// TIA Portal V20 export
// export: Created 2025-12-01T14:57:05.6941623Z, ExportSetting None, DisplayName Totally Integrated Automation Portal, DisplayVersion V20 Update 3, DisplayName TIA Portal Openness, DisplayVersion V20 Update 3, DisplayName TIA Portal Version Control Interface, DisplayVersion V20 Update 3, DisplayName STEP 7 Professional, DisplayVersion V20 Update 3, DisplayName STEP 7 Safety, DisplayVersion V20 Update 2, DisplayName WinCC Basic/Comfort/Advanced, DisplayVersion V20 Update 3, DisplayName WinCC Professional, DisplayVersion V20 Update 3, DisplayName WinCC Unified, DisplayVersion V20 Update 3
FUNCTION "FC876_BorrarEstructura" : Void   // FC876, LAD
TITLE = BorrarEstructura
{ S7_Optimized_Access := 'FALSE' }
AUTHOR : TRACKING
NAME : 20130301
VERSION : 3.0
// Borra un numero de bytes de un DB desde Offset que se indique
// stored: AutoNumber false, SetENOAutomatically false
   VAR_INPUT
      NumDB : Word;   // Numero del DB
      POffset : DWord;   // Puntero del Offset dento del DB
      NumBytes : UInt;   // Numero de Bytes que hay que borrar
   END_VAR
   VAR_TEMP
      Guardar_AR1 : DWord;
      Guardar_AR2 : DWord;
      PAny_DB : Any;
      ReturnValor : Int;
      Cero : Byte;
   END_VAR
BEGIN

NETWORK
TITLE = Inicializar Punteros Any
//////////////////////////////////////////////////////////////////////////////
//////////////////////////////////////////////////////////////////////////////
/// Tareas Iniciales

      TAR1  #Guardar_AR1;  // Guardar AR1 y AR2
      TAR2  #Guardar_AR2;


//////////////////////////////////////////////////////////////////////////////
//////////////////////////////////////////////////////////////////////////////
/// Puntero Any Origen

      LAR2  P##PAny_DB;  // - Any - DB de Origen
      L     B#16#10;  //   10H para S7
      T     LB [AR2, P#0.0];
      L     B#16#2;  //   Tipo de Datos (BYTE)
      T     LB [AR2, P#1.0];
      L     #NumBytes;  //   Cantidad de datos
      T     LW [AR2, P#2.0];
      L     #NumDB;  //   Numero de DB
      T     LW [AR2, P#4.0];
      L     #POffset;  //   Direccion de Inicio
      T     LD [AR2, P#6.0];
      L     B#16#84;  //   El Area de Memoria = DB (Nota: No 84)
      T     LB [AR2, P#6.0];


//////////////////////////////////////////////////////////////////////////////
//////////////////////////////////////////////////////////////////////////////
/// Tareas Finales

      LAR1  #Guardar_AR1;  // Recuperar AR1 y AR2
      LAR2  #Guardar_AR2;



NETWORK
TITLE = Borrado
//////////////////////////////////////////////////////////////////////////////
//////////////////////////////////////////////////////////////////////////////
/// Borrrado de los Datos

      L     0;
      T     #Cero;

      CALL  FILL
      ( BVAL    := #Cero,
        RET_VAL := #ReturnValor,
        BLK     := #PAny_DB
      );  // Inicializo las Entradas



END_FUNCTION
